TYPE
    CUBaseStatusInfo EXTENDS TcoCore.TcoStruct :
    STRUCT
     Mode                   : eCUMode;
     CurrentTaskDescription : STRING;
     CurrentUid             : INT;
     CurrentOperation       : STRING(255);
     CurrentCycleTime       : TIME;
	 AverageCycleTime       : TIME;
     CurrentIsInStepMode    : BOOL;
     CurrentCleanCycleTime  : TIME;
	 AverageCleanCycleTime  : TIME;
     State	                : eCUState;
     InSavingEnergy         : BOOL;
    END_STRUCT
END_TYPE

(* stored: Version 1.1.0.1
   DUT CUBaseStatusInfo: Id {0c2cb051-bd9e-41fb-9ccd-015b2464ed4a} *)
